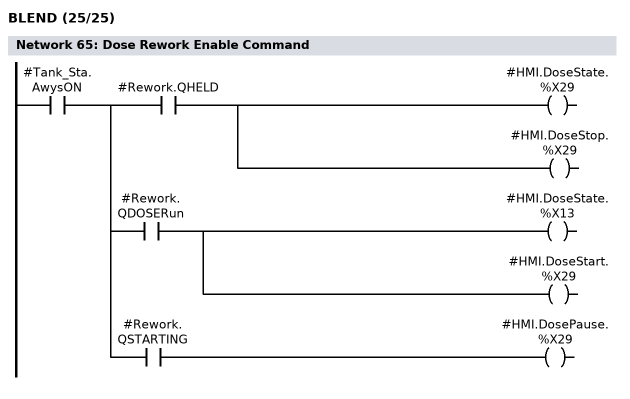
   RUNG wire#powerrail
      Contact( #Tank_Sta.AwysON )
      wire#w1
      Contact( #Rework.QHELD )
      wire#w2
      Coil( #HMI.DoseState.%X29 )
   END_RUNG
   RUNG wire#w2
      Coil( #HMI.DoseStop.%X29 )
   END_RUNG
   RUNG wire#w1
      Contact( #Rework.QDOSERun )
      wire#w3
      Coil( #HMI.DoseState.%X13 )
   END_RUNG
   RUNG wire#w3
      Coil( #HMI.DoseStart.%X29 )
   END_RUNG
   RUNG wire#w1
      Contact( #Rework.QSTARTING )
      Coil( #HMI.DosePause.%X29 )
   END_RUNG
   // the same network as SCL:
   #HMI.DoseState.%X29 := #Tank_Sta.AwysON AND #Rework.QHELD;
   #HMI.DoseStop.%X29 := #HMI.DoseState.%X29;
   #HMI.DoseState.%X13 := #Tank_Sta.AwysON AND #Rework.QDOSERun;
   #HMI.DoseStart.%X29 := #HMI.DoseState.%X13;
   #HMI.DosePause.%X29 := #Tank_Sta.AwysON AND #Rework.QSTARTING;
END_REGION
END_FUNCTION_BLOCK
